(* Logix 5000 project; controller Uidaho_Factory vendor 1 type 14 code 165 rev 38.11; software revision 38.00; part 2 of 3 *)
(* tags used below, declared in another part *)
   ESTOP : BOOL;
   HBW_Start : DINT;
   HBW_Step : DINT;
   HBW_X_Bound : DINT;
   HBW_X_Init : DINT;
   HBW_X_Offset : DINT;
   HBW_X_Position : DINT;
   HBW_Y_Bound : DINT;
   HBW_Y_Init : DINT;
   HBW_Y_Offset : DINT;
   HBW_Y_Position : DINT;
   MPO_start : DINT;
   Position : DINT;
   Start : DINT;
   X_Position_Return : DINT;
   Y_Position_Drop_off : DINT;
   Y_Position_DropOff_At_Rack : DINT;
   Y_Position_Pick_Up : DINT;
   Y_Position_Return : DINT;
   Encoder_Counters_1X : COUNTER[10];
   Encoder_Counters_4X : COUNTER[10];
   I_O_Counter : COUNTER[20];
   PWM_Outputs : PWM_Out[20];
   Slot_1_Faulted : DINT;
   Slot_2_Faulted : DINT;
   Slot_3_Faulted : DINT;
   Slot_4_Faulted : DINT;
   Slot_5_Faulted : DINT;
   Slot_6_Faulted : DINT;
   Slot_7_Faulted : DINT;
   Slot_9_Faulted : DINT;
(* MainProgram, continued *)

ROUTINE HBW_Controller   (* ladder *)
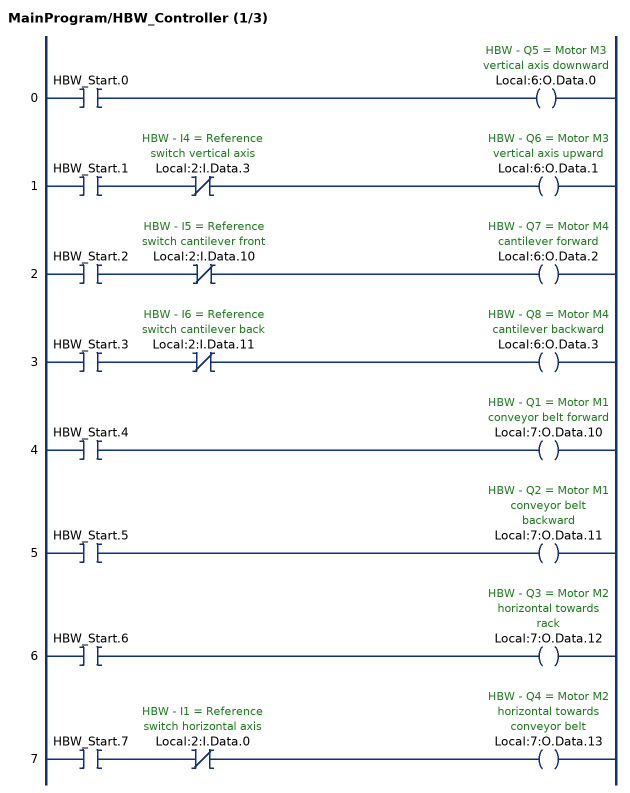
   0: XIC(HBW_Start.0)OTE(Local:6:O.Data.0);
   1: XIC(HBW_Start.1)XIO(Local:2:I.Data.3)OTE(Local:6:O.Data.1);
   2: XIC(HBW_Start.2)XIO(Local:2:I.Data.10)OTE(Local:6:O.Data.2);
   3: XIC(HBW_Start.3)XIO(Local:2:I.Data.11)OTE(Local:6:O.Data.3);
   4: XIC(HBW_Start.4)OTE(Local:7:O.Data.10);
   5: XIC(HBW_Start.5)OTE(Local:7:O.Data.11);
   6: XIC(HBW_Start.6)OTE(Local:7:O.Data.12);
   7: XIC(HBW_Start.7)XIO(Local:2:I.Data.0)OTE(Local:7:O.Data.13);
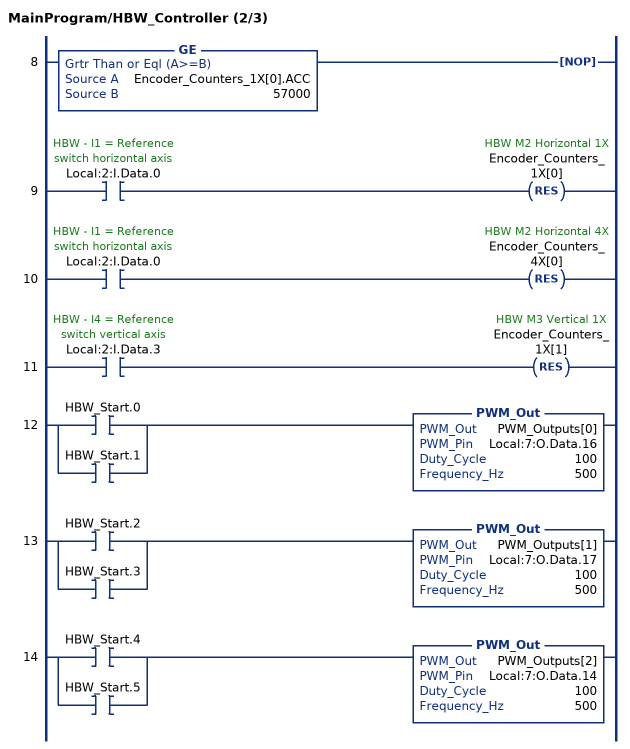
   8: GE(Encoder_Counters_1X[0].ACC,57000)NOP();
   9: XIC(Local:2:I.Data.0)RES(Encoder_Counters_1X[0]);
   10: XIC(Local:2:I.Data.0)RES(Encoder_Counters_4X[0]);
   11: XIC(Local:2:I.Data.3)RES(Encoder_Counters_1X[1]);
   12: [XIC(HBW_Start.0) ,XIC(HBW_Start.1) ]PWM_Out(PWM_Outputs[0],Local:7:O.Data.16,100,500);
   13: [XIC(HBW_Start.2) ,XIC(HBW_Start.3) ]PWM_Out(PWM_Outputs[1],Local:7:O.Data.17,100,500);
   14: [XIC(HBW_Start.4) ,XIC(HBW_Start.5) ]PWM_Out(PWM_Outputs[2],Local:7:O.Data.14,100,500);
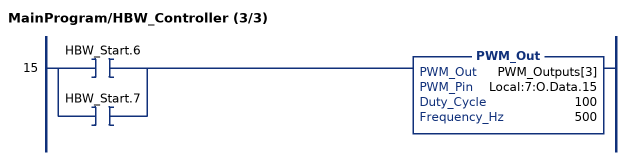
   15: [XIC(HBW_Start.6) ,XIC(HBW_Start.7) ]PWM_Out(PWM_Outputs[3],Local:7:O.Data.15,100,500);
END_ROUTINE

ROUTINE HBW_Sequencer   (* ladder *)
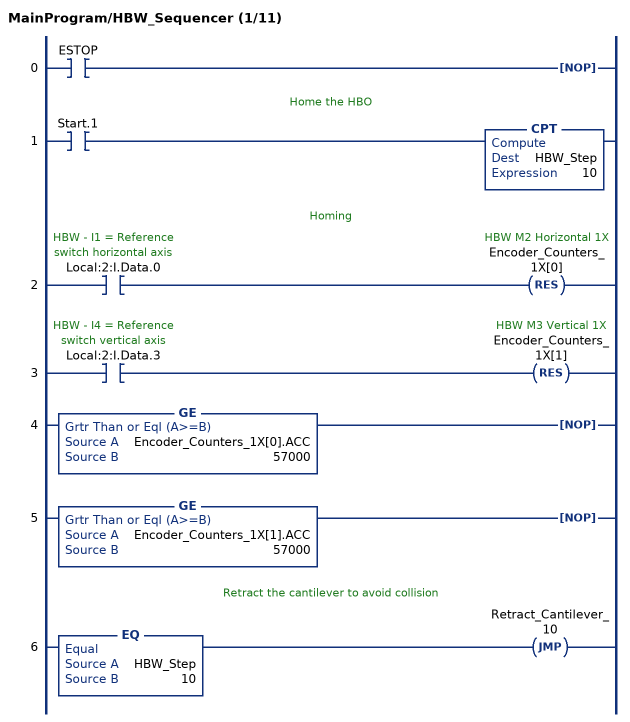
   0: XIC(ESTOP)NOP();
   // Home the HBO
   1: XIC(Start.1)CPT(HBW_Step,10);
   // Homing
   2: XIC(Local:2:I.Data.0)RES(Encoder_Counters_1X[0]);
   3: XIC(Local:2:I.Data.3)RES(Encoder_Counters_1X[1]);
   4: GE(Encoder_Counters_1X[0].ACC,57000)NOP();
   5: GE(Encoder_Counters_1X[1].ACC,57000)NOP();
   // Retract the cantilever to avoid collision
   6: EQ(HBW_Step,10)JMP(Retract_Cantilever_10);
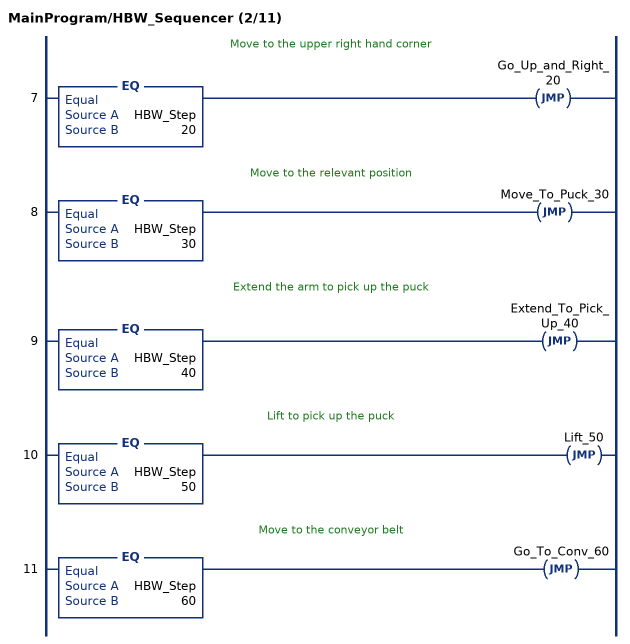
   // Move to the upper right hand corner
   7: EQ(HBW_Step,20)JMP(Go_Up_and_Right_20);
   // Move to the relevant position
   8: EQ(HBW_Step,30)JMP(Move_To_Puck_30);
   // Extend the arm to pick up the puck
   9: EQ(HBW_Step,40)JMP(Extend_To_Pick_Up_40);
   // Lift to pick up the puck
   10: EQ(HBW_Step,50)JMP(Lift_50);
   // Move to the conveyor belt
   11: EQ(HBW_Step,60)JMP(Go_To_Conv_60);
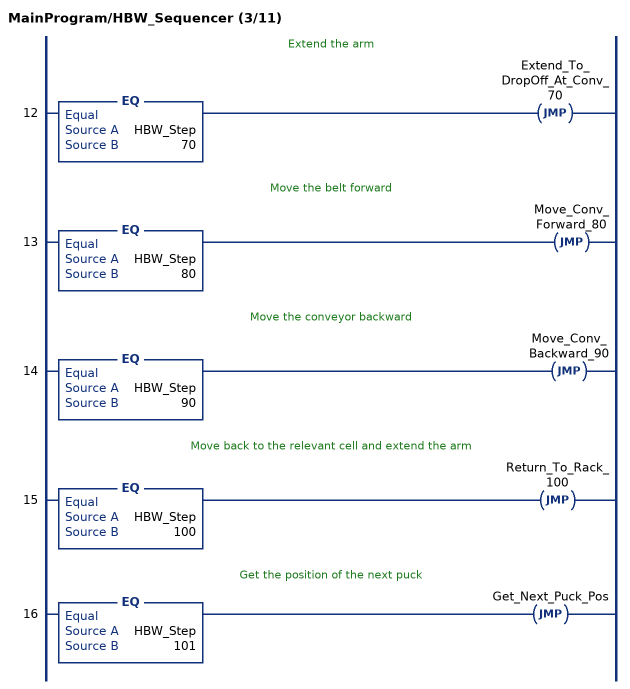
   // Extend the arm
   12: EQ(HBW_Step,70)JMP(Extend_To_DropOff_At_Conv_70);
   // Move the belt forward
   13: EQ(HBW_Step,80)JMP(Move_Conv_Forward_80);
   // Move the conveyor backward
   14: EQ(HBW_Step,90)JMP(Move_Conv_Backward_90);
   // Move back to the relevant cell and extend the arm
   15: EQ(HBW_Step,100)JMP(Return_To_Rack_100);
   // Get the position of the next puck
   16: EQ(HBW_Step,101)JMP(Get_Next_Puck_Pos);
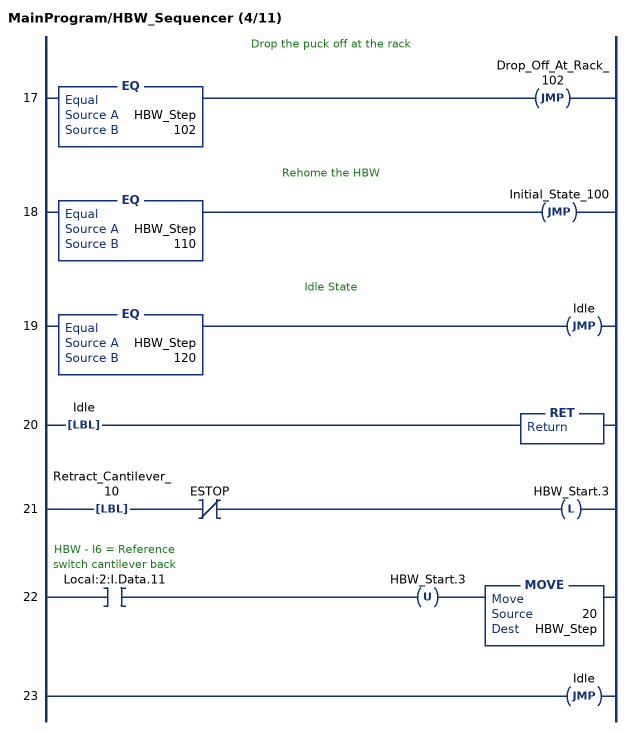
   // Drop the puck off at the rack
   17: EQ(HBW_Step,102)JMP(Drop_Off_At_Rack_102);
   // Rehome the HBW
   18: EQ(HBW_Step,110)JMP(Initial_State_100);
   // Idle State
   19: EQ(HBW_Step,120)JMP(Idle);
   20: LBL(Idle)RET();
   21: LBL(Retract_Cantilever_10)XIO(ESTOP)OTL(HBW_Start.3);
   22: XIC(Local:2:I.Data.11)OTU(HBW_Start.3)MOVE(20,HBW_Step);
   23: JMP(Idle);
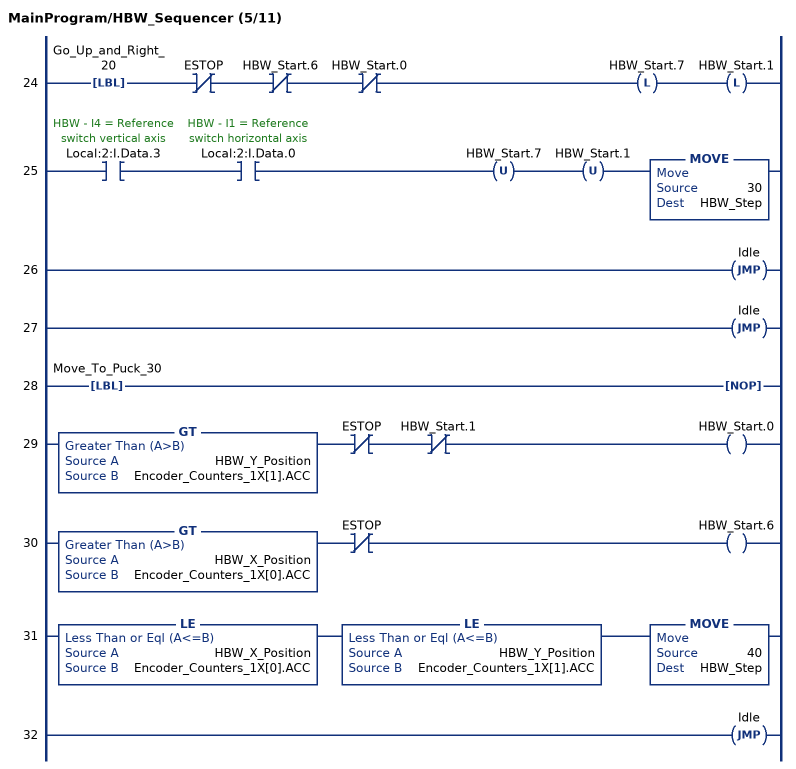
   24: LBL(Go_Up_and_Right_20)XIO(ESTOP)XIO(HBW_Start.6)XIO(HBW_Start.0)OTL(HBW_Start.7)OTL(HBW_Start.1);
   25: XIC(Local:2:I.Data.3)XIC(Local:2:I.Data.0)OTU(HBW_Start.7)OTU(HBW_Start.1)MOVE(30,HBW_Step);
   26: JMP(Idle);
   27: JMP(Idle);
   28: LBL(Move_To_Puck_30)NOP();
   29: GT(HBW_Y_Position,Encoder_Counters_1X[1].ACC)XIO(ESTOP)XIO(HBW_Start.1)OTE(HBW_Start.0);
   30: GT(HBW_X_Position,Encoder_Counters_1X[0].ACC)XIO(ESTOP)OTE(HBW_Start.6);
   31: LE(HBW_X_Position,Encoder_Counters_1X[0].ACC)LE(HBW_Y_Position,Encoder_Counters_1X[1].ACC)MOVE(40,HBW_Step);
   32: JMP(Idle);
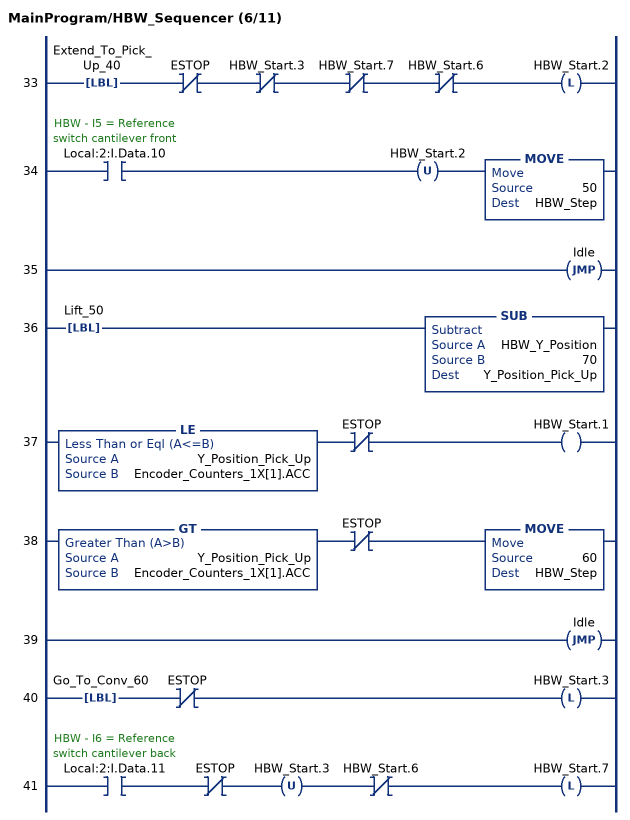
   33: LBL(Extend_To_Pick_Up_40)XIO(ESTOP)XIO(HBW_Start.3)XIO(HBW_Start.7)XIO(HBW_Start.6)OTL(HBW_Start.2);
   34: XIC(Local:2:I.Data.10)OTU(HBW_Start.2)MOVE(50,HBW_Step);
   35: JMP(Idle);
   36: LBL(Lift_50)SUB(HBW_Y_Position,70,Y_Position_Pick_Up);
   37: LE(Y_Position_Pick_Up,Encoder_Counters_1X[1].ACC)XIO(ESTOP)OTE(HBW_Start.1);
   38: GT(Y_Position_Pick_Up,Encoder_Counters_1X[1].ACC)XIO(ESTOP)MOVE(60,HBW_Step);
   39: JMP(Idle);
   40: LBL(Go_To_Conv_60)XIO(ESTOP)OTL(HBW_Start.3);
   41: XIC(Local:2:I.Data.11)XIO(ESTOP)OTU(HBW_Start.3)XIO(HBW_Start.6)OTL(HBW_Start.7);
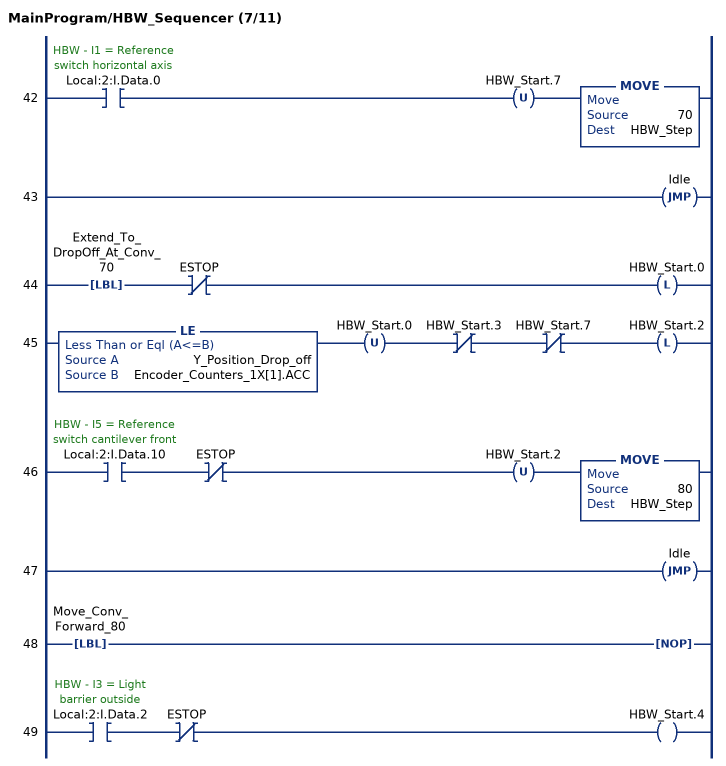
   42: XIC(Local:2:I.Data.0)OTU(HBW_Start.7)MOVE(70,HBW_Step);
   43: JMP(Idle);
   44: LBL(Extend_To_DropOff_At_Conv_70)XIO(ESTOP)OTL(HBW_Start.0);
   45: LE(Y_Position_Drop_off,Encoder_Counters_1X[1].ACC)OTU(HBW_Start.0)XIO(HBW_Start.3)XIO(HBW_Start.7)OTL(HBW_Start.2);
   46: XIC(Local:2:I.Data.10)XIO(ESTOP)OTU(HBW_Start.2)MOVE(80,HBW_Step);
   47: JMP(Idle);
   48: LBL(Move_Conv_Forward_80)NOP();
   49: XIC(Local:2:I.Data.2)XIO(ESTOP)OTE(HBW_Start.4);
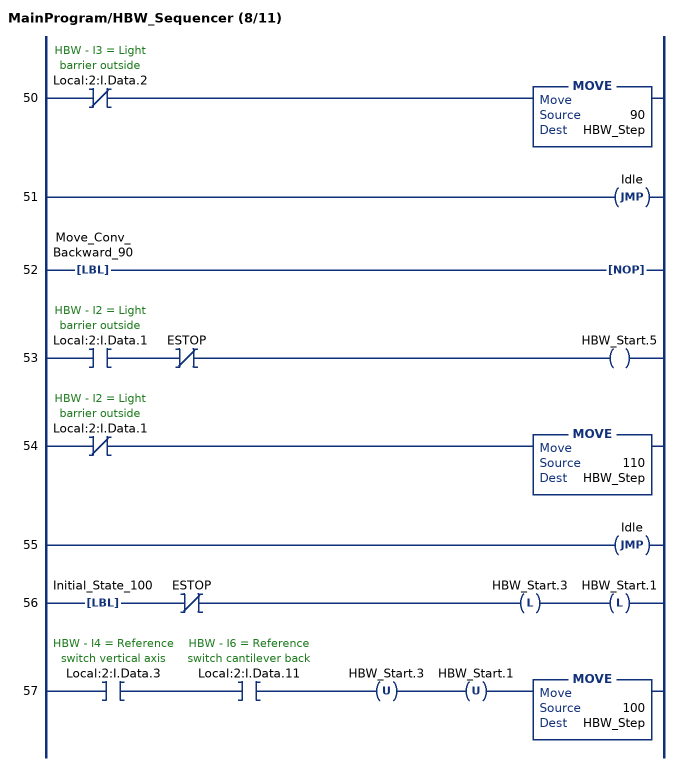
   50: XIO(Local:2:I.Data.2)MOVE(90,HBW_Step);
   51: JMP(Idle);
   52: LBL(Move_Conv_Backward_90)NOP();
   53: XIC(Local:2:I.Data.1)XIO(ESTOP)OTE(HBW_Start.5);
   54: XIO(Local:2:I.Data.1)MOVE(110,HBW_Step);
   55: JMP(Idle);
   56: LBL(Initial_State_100)XIO(ESTOP)OTL(HBW_Start.3)OTL(HBW_Start.1);
   57: XIC(Local:2:I.Data.3)XIC(Local:2:I.Data.11)OTU(HBW_Start.3)OTU(HBW_Start.1)MOVE(100,HBW_Step);
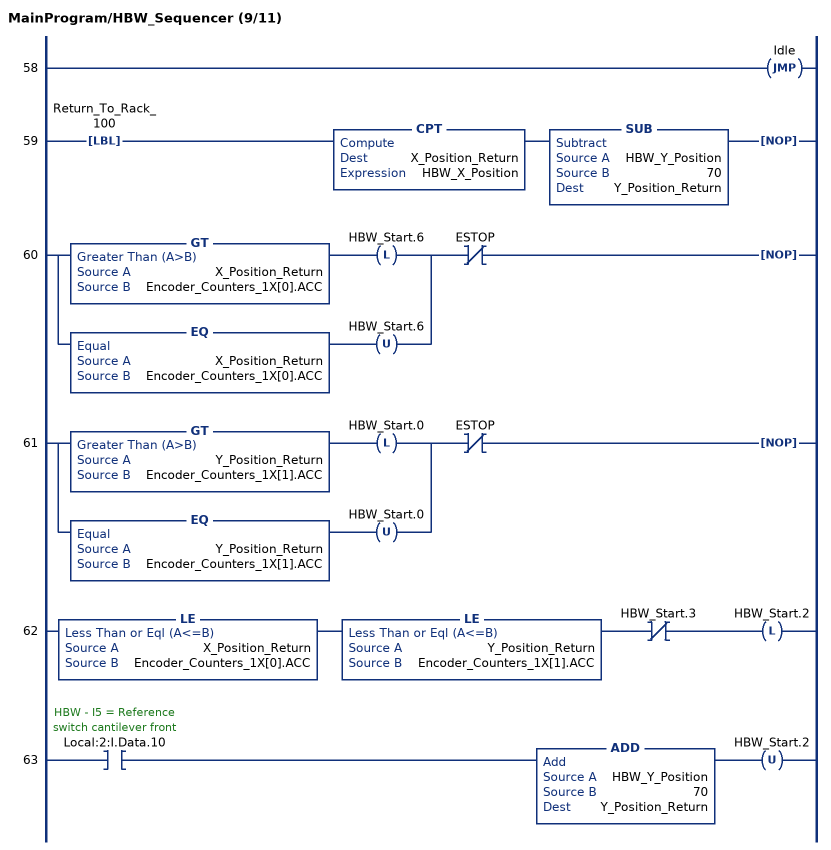
   58: JMP(Idle);
   59: LBL(Return_To_Rack_100)CPT(X_Position_Return,HBW_X_Position)SUB(HBW_Y_Position,70,Y_Position_Return)NOP();
   60: [GT(X_Position_Return,Encoder_Counters_1X[0].ACC) OTL(HBW_Start.6) ,EQ(X_Position_Return,Encoder_Counters_1X[0].ACC) OTU(HBW_Start.6) ]XIO(ESTOP)NOP();
   61: [GT(Y_Position_Return,Encoder_Counters_1X[1].ACC) OTL(HBW_Start.0) ,EQ(Y_Position_Return,Encoder_Counters_1X[1].ACC) OTU(HBW_Start.0) ]XIO(ESTOP)NOP();
   62: LE(X_Position_Return,Encoder_Counters_1X[0].ACC)LE(Y_Position_Return,Encoder_Counters_1X[1].ACC)XIO(HBW_Start.3)OTL(HBW_Start.2);
   63: XIC(Local:2:I.Data.10)ADD(HBW_Y_Position,70,Y_Position_Return)OTU(HBW_Start.2);
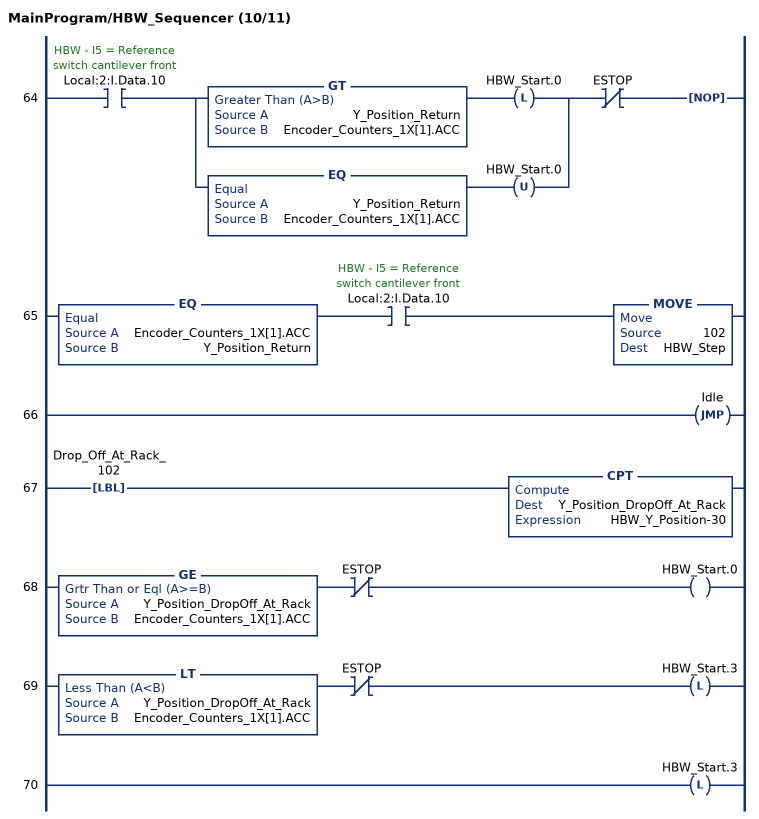
   64: XIC(Local:2:I.Data.10)[GT(Y_Position_Return,Encoder_Counters_1X[1].ACC) OTL(HBW_Start.0) ,EQ(Y_Position_Return,Encoder_Counters_1X[1].ACC) OTU(HBW_Start.0) ]XIO(ESTOP)NOP();
   65: EQ(Encoder_Counters_1X[1].ACC,Y_Position_Return)XIC(Local:2:I.Data.10)MOVE(102,HBW_Step);
   66: JMP(Idle);
   67: LBL(Drop_Off_At_Rack_102)CPT(Y_Position_DropOff_At_Rack,HBW_Y_Position-30);
   68: GE(Y_Position_DropOff_At_Rack,Encoder_Counters_1X[1].ACC)XIO(ESTOP)OTE(HBW_Start.0);
   69: LT(Y_Position_DropOff_At_Rack,Encoder_Counters_1X[1].ACC)XIO(ESTOP)OTL(HBW_Start.3);
   70: OTL(HBW_Start.3);
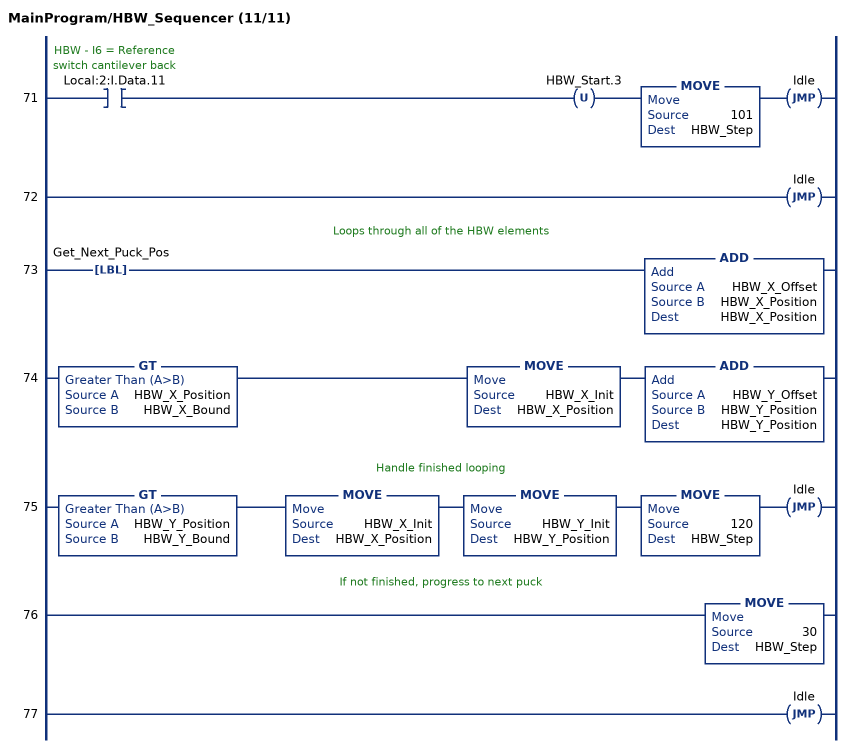
   71: XIC(Local:2:I.Data.11)OTU(HBW_Start.3)MOVE(101,HBW_Step)JMP(Idle);
   72: JMP(Idle);
   // Loops through all of the HBW elements
   73: LBL(Get_Next_Puck_Pos)ADD(HBW_X_Offset,HBW_X_Position,HBW_X_Position);
   74: GT(HBW_X_Position,HBW_X_Bound)MOVE(HBW_X_Init,HBW_X_Position)ADD(HBW_Y_Offset,HBW_Y_Position,HBW_Y_Position);
   // Handle finished looping
   75: GT(HBW_Y_Position,HBW_Y_Bound)MOVE(HBW_X_Init,HBW_X_Position)MOVE(HBW_Y_Init,HBW_Y_Position)MOVE(120,HBW_Step)JMP(Idle);
   // If not finished, progress to next puck
   76: MOVE(30,HBW_Step);
   77: JMP(Idle);
END_ROUTINE

ROUTINE MainRoutine   (* ladder *)
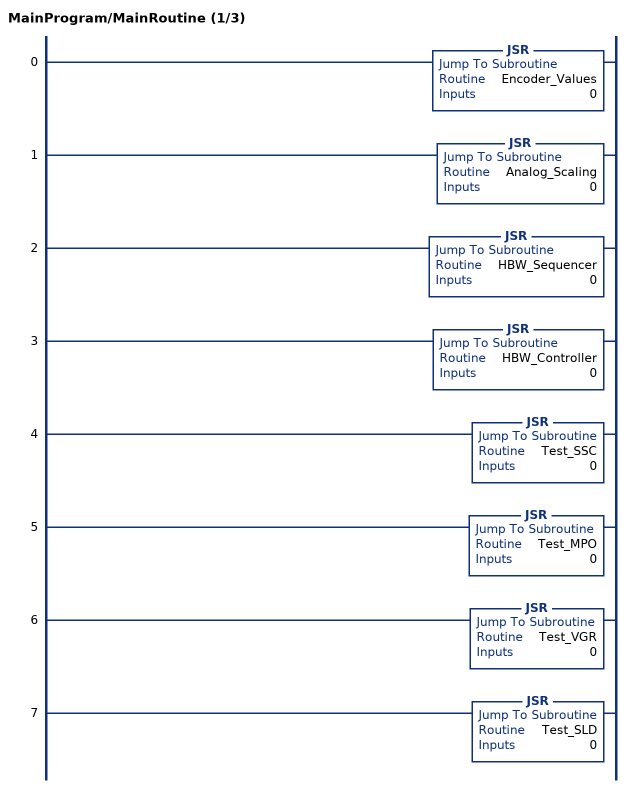
   0: JSR(Encoder_Values,0);
   1: JSR(Analog_Scaling,0);
   2: JSR(HBW_Sequencer,0);
   3: JSR(HBW_Controller,0);
   4: JSR(Test_SSC,0);
   5: JSR(Test_MPO,0);
   6: JSR(Test_VGR,0);
   7: JSR(Test_SLD,0);
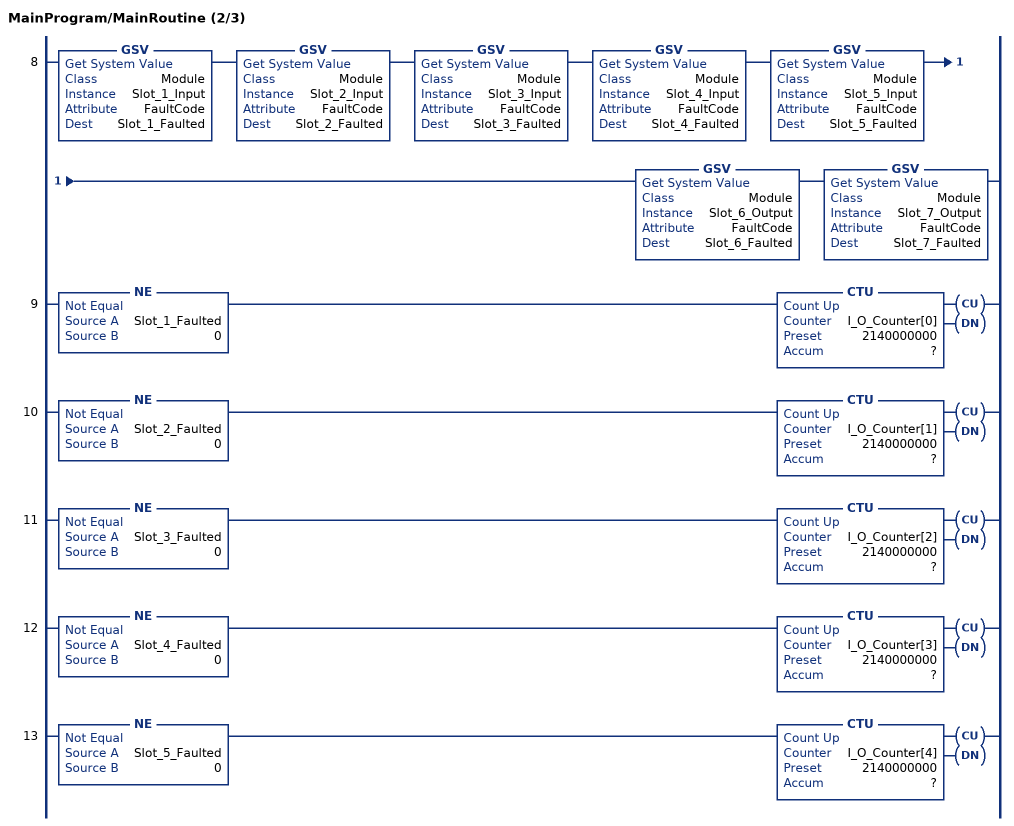
   8: GSV(Module,Slot_1_Input,FaultCode,Slot_1_Faulted)GSV(Module,Slot_2_Input,FaultCode,Slot_2_Faulted)GSV(Module,Slot_3_Input,FaultCode,Slot_3_Faulted)GSV(Module,Slot_4_Input,FaultCode,Slot_4_Faulted)GSV(Module,Slot_5_Input,FaultCode,Slot_5_Faulted)GSV(Module,Slot_6_Output,FaultCode,Slot_6_Faulted)GSV(Module,Slot_7_Output,FaultCode,Slot_7_Faulted);
   9: NE(Slot_1_Faulted,0)CTU(I_O_Counter[0],?,?);
   10: NE(Slot_2_Faulted,0)CTU(I_O_Counter[1],?,?);
   11: NE(Slot_3_Faulted,0)CTU(I_O_Counter[2],?,?);
   12: NE(Slot_4_Faulted,0)CTU(I_O_Counter[3],?,?);
   13: NE(Slot_5_Faulted,0)CTU(I_O_Counter[4],?,?);
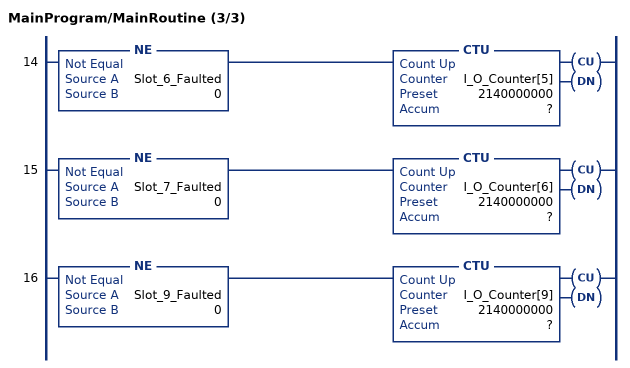
   14: NE(Slot_6_Faulted,0)CTU(I_O_Counter[5],?,?);
   15: NE(Slot_7_Faulted,0)CTU(I_O_Counter[6],?,?);
   16: NE(Slot_9_Faulted,0)CTU(I_O_Counter[9],?,?);
END_ROUTINE

ROUTINE Test_MPO   (* ladder *)
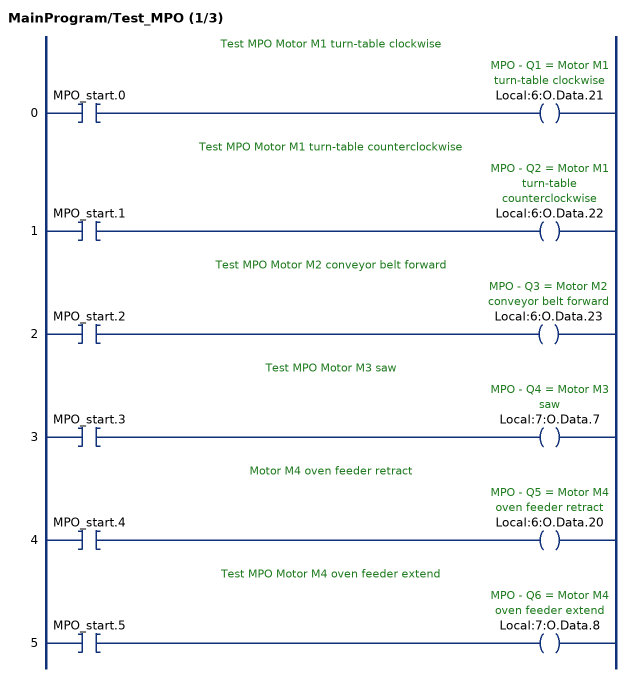
   // Test MPO Motor M1 turn-table clockwise
   0: XIC(MPO_start.0)OTE(Local:6:O.Data.21);
   // Test MPO Motor M1 turn-table counterclockwise
   1: XIC(MPO_start.1)OTE(Local:6:O.Data.22);
   // Test MPO Motor M2 conveyor belt forward
   2: XIC(MPO_start.2)OTE(Local:6:O.Data.23);
   // Test MPO Motor M3 saw
   3: XIC(MPO_start.3)OTE(Local:7:O.Data.7);
   // Motor M4 oven feeder retract
   4: XIC(MPO_start.4)OTE(Local:6:O.Data.20);
   // Test MPO Motor M4 oven feeder extend
   5: XIC(MPO_start.5)OTE(Local:7:O.Data.8);
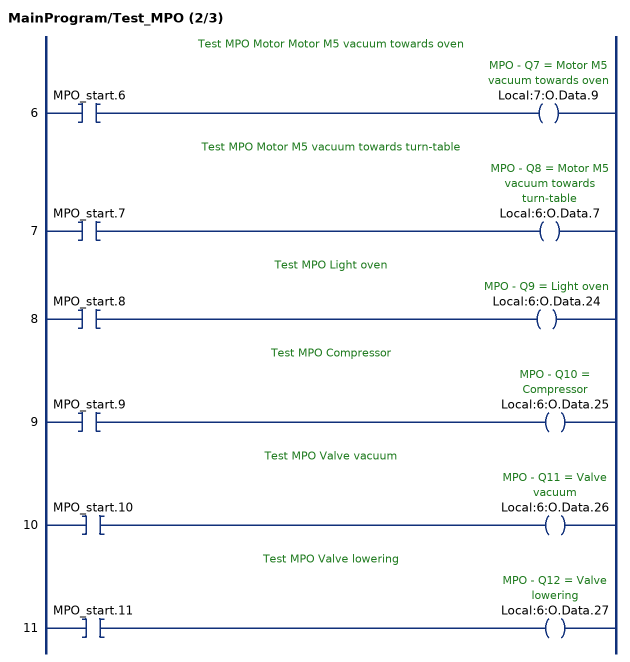
   // Test MPO Motor Motor M5 vacuum towards oven
   6: XIC(MPO_start.6)OTE(Local:7:O.Data.9);
   // Test MPO Motor M5 vacuum towards turn-table
   7: XIC(MPO_start.7)OTE(Local:6:O.Data.7);
   // Test MPO Light oven
   8: XIC(MPO_start.8)OTE(Local:6:O.Data.24);
   // Test MPO Compressor
   9: XIC(MPO_start.9)OTE(Local:6:O.Data.25);
   // Test MPO Valve vacuum
   10: XIC(MPO_start.10)OTE(Local:6:O.Data.26);
   // Test MPO Valve lowering
   11: XIC(MPO_start.11)OTE(Local:6:O.Data.27);
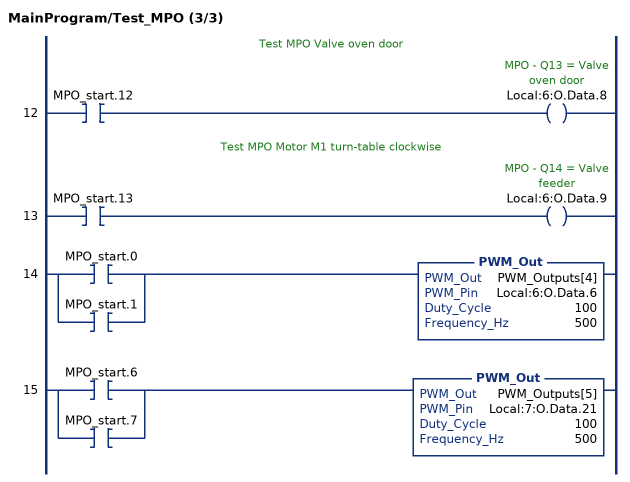
   // Test MPO Valve oven door
   12: XIC(MPO_start.12)OTE(Local:6:O.Data.8);
   // Test MPO Motor M1 turn-table clockwise
   13: XIC(MPO_start.13)OTE(Local:6:O.Data.9);
   14: [XIC(MPO_start.0) ,XIC(MPO_start.1) ]PWM_Out(PWM_Outputs[4],Local:6:O.Data.6,100,500);
   15: [XIC(MPO_start.6) ,XIC(MPO_start.7) ]PWM_Out(PWM_Outputs[5],Local:7:O.Data.21,100,500);
END_ROUTINE
